// TIA Portal V20 export
FUNCTION_BLOCK "Sequence_1_VisionUnit"   // FB160, LAD
TITLE = Sequence
// Sequence template programmend in ladder logic
// stored: IsIECCheckEnabled true, MemoryReserve 100, Namespace Unit1.Em6, SetENOAutomatically true
   VAR_OUTPUT
      safeState : Bool;
   END_VAR
   VAR
      instSequenceLADControl { ExternalWritable := 'False'} : "LAF_ControlLadSequence";
      instSequenceLADStatus { ExternalWritable := 'False'} : "LAF_StatusLadSequence";
      statPulse { ExternalWritable := 'False'} : Array[0..999] of Bool;
      statTonTimer { ExternalWritable := 'False'} : Array[0..1999] of TON_TIME;
   END_VAR
   VAR_TEMP
      tempCustomerAction : Bool;   // Placeholder for possible actions
      tempDo_nothing_and_wait_for_init : Bool;   // Placeholder for doing nothing
      tempSafeStateCondition : Bool;   // Temp Condition for the equipment module to be in a safe state
   END_VAR
   VAR CONSTANT
      STEP_IDLE : DInt := 1;   // Idle Step
      JOB_1_STEP_01 : DInt := 101;
      JOB_1_STEP_11 : DInt := 111;
      JOB_1_STEP_21 : DInt := 121;
      JOB_1_STEP_31 : DInt := 131;
      JOB_1_STEP_91 : DInt := 191;
      JOB_2_STEP_01 : DInt := 201;
      JOB_2_STEP_11 : DInt := 211;
      JOB_2_STEP_91 : DInt := 291;
      JOB_3_STEP_01 : DInt := 301;
      JOB_3_STEP_11 : DInt := 311;
      JOB_3_STEP_91 : DInt := 391;
      JOB_10_STEP_01 : DInt := 1001;
      JOB_10_STEP_11 : DInt := 1011;
      JOB_10_STEP_21 : DInt := 1021;
      JOB_10_STEP_31 : DInt := 1031;
      JOB_10_STEP_41 : DInt := 1041;
      JOB_10_STEP_51 : DInt := 1051;
      JOB_10_STEP_61 : DInt := 1061;
      JOB_10_STEP_71 : DInt := 1071;
      JOB_10_STEP_81 : DInt := 1081;
      JOB_10_STEP_91 : DInt := 1091;
      STEP_IMMEDIATE_STOP : DInt := 9001;   // Step executed when an immediate stop command is triggered for the sequence (i.e. when unit is in state aborting)
      SeqDelayTime : Time := T#100ms;
      SeqNoDelayTime : Time;
      TRUE : Bool := TRUE;
      FALSE : Bool := FALSE;
      VisionUnitAxisZHomePos : SInt := 0;
      VisionUnitAxisZVisionPos : SInt := 1;
   END_VAR
   VAR_TEMP   // added for the SCL form of the ladder/FBD networks
      _w1 : Bool;
      _w2 : Bool;
   END_VAR
BEGIN

REGION Network 1: BLOCK INFO HEADER
   // (company) / (C) Copyright (year)
   // ---------------------------------------------------------------------------------
   // Title:                             (Title of this block)
   // Comment/Function: (that is implemented in the block)
   // Library/Family:           (that the source is dedicated to)
   // Author:                        (department / person in charge / contact)
   // Target System:          (test system with FW version)
   // Engineering:              TIA Portal (SW version)
   // Restrictions:               (OB types, etc.)
   // Requirements:           (hardware, technological package, etc.)
   // ---------------------------------------------------------------------------------
   // Change log table:
   // Version          | Date             | Signature      | Expert in charge  | Changes applied ------------------------|----------------------|-------------------------|--------------------------------|-----------------------
   // 001.000.000 | yyyy-mm-dd | 0x00000000 | (name of expert) | First released version
END_REGION

REGION Network 2: DESCRIPTION
   // This is a template block provided by the Automation Framework. It can be used to create an own project.
   // The Block Info Header is prepared to put in your own data.
   // Description of the block could be added here and the docu created by Code2Docu.
END_REGION

REGION Network 3: *************** CONTROL **********************
END_REGION

REGION Network 4: Sequence Control
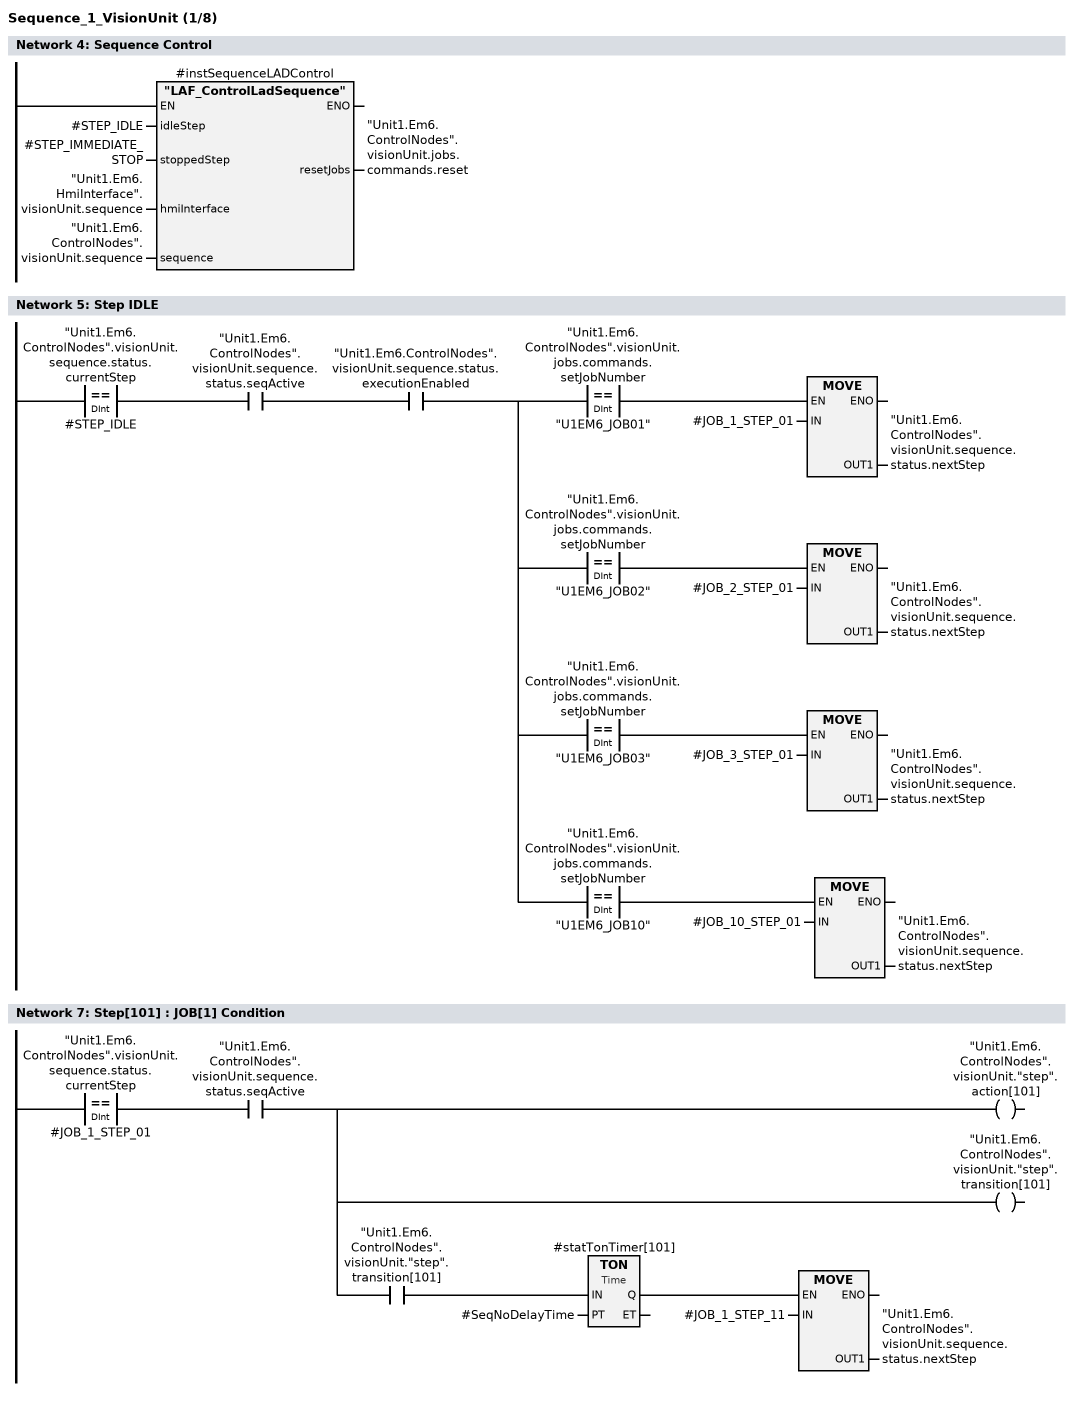
   RUNG wire#powerrail
      #instSequenceLADControl(idleStep := #STEP_IDLE, stoppedStep := #STEP_IMMEDIATE_STOP, hmiInterface := "Unit1.Em6.HmiInterface".visionUnit.sequence, sequence := "Unit1.Em6.ControlNodes".visionUnit.sequence, resetJobs => "Unit1.Em6.ControlNodes".visionUnit.jobs.commands.reset)
   END_RUNG
   // the same network as SCL:
   #instSequenceLADControl(idleStep := #STEP_IDLE,   // "LAF_ControlLadSequence"
                           stoppedStep := #STEP_IMMEDIATE_STOP,
                           hmiInterface := "Unit1.Em6.HmiInterface".visionUnit.sequence,
                           sequence := "Unit1.Em6.ControlNodes".visionUnit.sequence,
                           resetJobs => "Unit1.Em6.ControlNodes".visionUnit.jobs.commands.reset);
END_REGION

REGION Network 5: Step IDLE
   RUNG wire#powerrail
      { S7_Templates := "SrcType := DInt" } EQ_Contact(in1 := "Unit1.Em6.ControlNodes".visionUnit.sequence.status.currentStep, in2 := #STEP_IDLE)
      Contact( "Unit1.Em6.ControlNodes".visionUnit.sequence.status.seqActive )
      Contact( "Unit1.Em6.ControlNodes".visionUnit.sequence.status.executionEnabled )
      wire#w1
      { S7_Templates := "SrcType := DInt" } EQ_Contact(in1 := "Unit1.Em6.ControlNodes".visionUnit.jobs.commands.setJobNumber, in2 := "U1EM6_JOB01")
      Move(in := #JOB_1_STEP_01, out1 => "Unit1.Em6.ControlNodes".visionUnit.sequence.status.nextStep)
   END_RUNG
   RUNG wire#w1
      { S7_Templates := "SrcType := DInt" } EQ_Contact(in1 := "Unit1.Em6.ControlNodes".visionUnit.jobs.commands.setJobNumber, in2 := "U1EM6_JOB02")
      Move(in := #JOB_2_STEP_01, out1 => "Unit1.Em6.ControlNodes".visionUnit.sequence.status.nextStep)
   END_RUNG
   RUNG wire#w1
      { S7_Templates := "SrcType := DInt" } EQ_Contact(in1 := "Unit1.Em6.ControlNodes".visionUnit.jobs.commands.setJobNumber, in2 := "U1EM6_JOB03")
      Move(in := #JOB_3_STEP_01, out1 => "Unit1.Em6.ControlNodes".visionUnit.sequence.status.nextStep)
   END_RUNG
   RUNG wire#w1
      { S7_Templates := "SrcType := DInt" } EQ_Contact(in1 := "Unit1.Em6.ControlNodes".visionUnit.jobs.commands.setJobNumber, in2 := "U1EM6_JOB10")
      Move(in := #JOB_10_STEP_01, out1 => "Unit1.Em6.ControlNodes".visionUnit.sequence.status.nextStep)
   END_RUNG
   // the same network as SCL:
   #_w1 := ("Unit1.Em6.ControlNodes".visionUnit.sequence.status.currentStep = #STEP_IDLE) AND "Unit1.Em6.ControlNodes".visionUnit.sequence.status.seqActive AND "Unit1.Em6.ControlNodes".visionUnit.sequence.status.executionEnabled;
   IF #_w1 AND ("Unit1.Em6.ControlNodes".visionUnit.jobs.commands.setJobNumber = "U1EM6_JOB01") THEN
       "Unit1.Em6.ControlNodes".visionUnit.sequence.status.nextStep := #JOB_1_STEP_01;
   END_IF;
   IF #_w1 AND ("Unit1.Em6.ControlNodes".visionUnit.jobs.commands.setJobNumber = "U1EM6_JOB02") THEN
       "Unit1.Em6.ControlNodes".visionUnit.sequence.status.nextStep := #JOB_2_STEP_01;
   END_IF;
   IF #_w1 AND ("Unit1.Em6.ControlNodes".visionUnit.jobs.commands.setJobNumber = "U1EM6_JOB03") THEN
       "Unit1.Em6.ControlNodes".visionUnit.sequence.status.nextStep := #JOB_3_STEP_01;
   END_IF;
   IF #_w1 AND ("Unit1.Em6.ControlNodes".visionUnit.jobs.commands.setJobNumber = "U1EM6_JOB10") THEN
       "Unit1.Em6.ControlNodes".visionUnit.sequence.status.nextStep := #JOB_10_STEP_01;
   END_IF;
END_REGION

REGION Network 6: *************** JOB 1 EM READY *************************
END_REGION

REGION Network 7: Step[101] : JOB[1] Condition
   RUNG wire#powerrail
      { S7_Templates := "SrcType := DInt" } EQ_Contact(in1 := "Unit1.Em6.ControlNodes".visionUnit.sequence.status.currentStep, in2 := #JOB_1_STEP_01)
      Contact( "Unit1.Em6.ControlNodes".visionUnit.sequence.status.seqActive )
      wire#w1
      Coil( "Unit1.Em6.ControlNodes".visionUnit."step".action[101] )
   END_RUNG
   RUNG wire#w1
      Coil( "Unit1.Em6.ControlNodes".visionUnit."step".transition[101] )
   END_RUNG
   RUNG wire#w1
      Contact( "Unit1.Em6.ControlNodes".visionUnit."step".transition[101] )
      { S7_Templates := "time_type := Time" } #statTonTimer[101].TON(pt := #SeqNoDelayTime, et =>)
      Move(in := #JOB_1_STEP_11, out1 => "Unit1.Em6.ControlNodes".visionUnit.sequence.status.nextStep)
   END_RUNG
   // the same network as SCL:
   "Unit1.Em6.ControlNodes".visionUnit."step".action[101] := ("Unit1.Em6.ControlNodes".visionUnit.sequence.status.currentStep = #JOB_1_STEP_01) AND "Unit1.Em6.ControlNodes".visionUnit.sequence.status.seqActive;
   "Unit1.Em6.ControlNodes".visionUnit."step".transition[101] := ("Unit1.Em6.ControlNodes".visionUnit.sequence.status.currentStep = #JOB_1_STEP_01) AND "Unit1.Em6.ControlNodes".visionUnit.sequence.status.seqActive;
   #statTonTimer[101].TON(IN := ("Unit1.Em6.ControlNodes".visionUnit.sequence.status.currentStep = #JOB_1_STEP_01) AND "Unit1.Em6.ControlNodes".visionUnit.sequence.status.seqActive AND "Unit1.Em6.ControlNodes".visionUnit."step".transition[101],
                          PT := #SeqNoDelayTime);
   IF #statTonTimer[101].Q THEN
       "Unit1.Em6.ControlNodes".visionUnit.sequence.status.nextStep := #JOB_1_STEP_11;
   END_IF;
END_REGION

REGION Network 8: Step[111] : Vision Unit AxisZ Homed Check
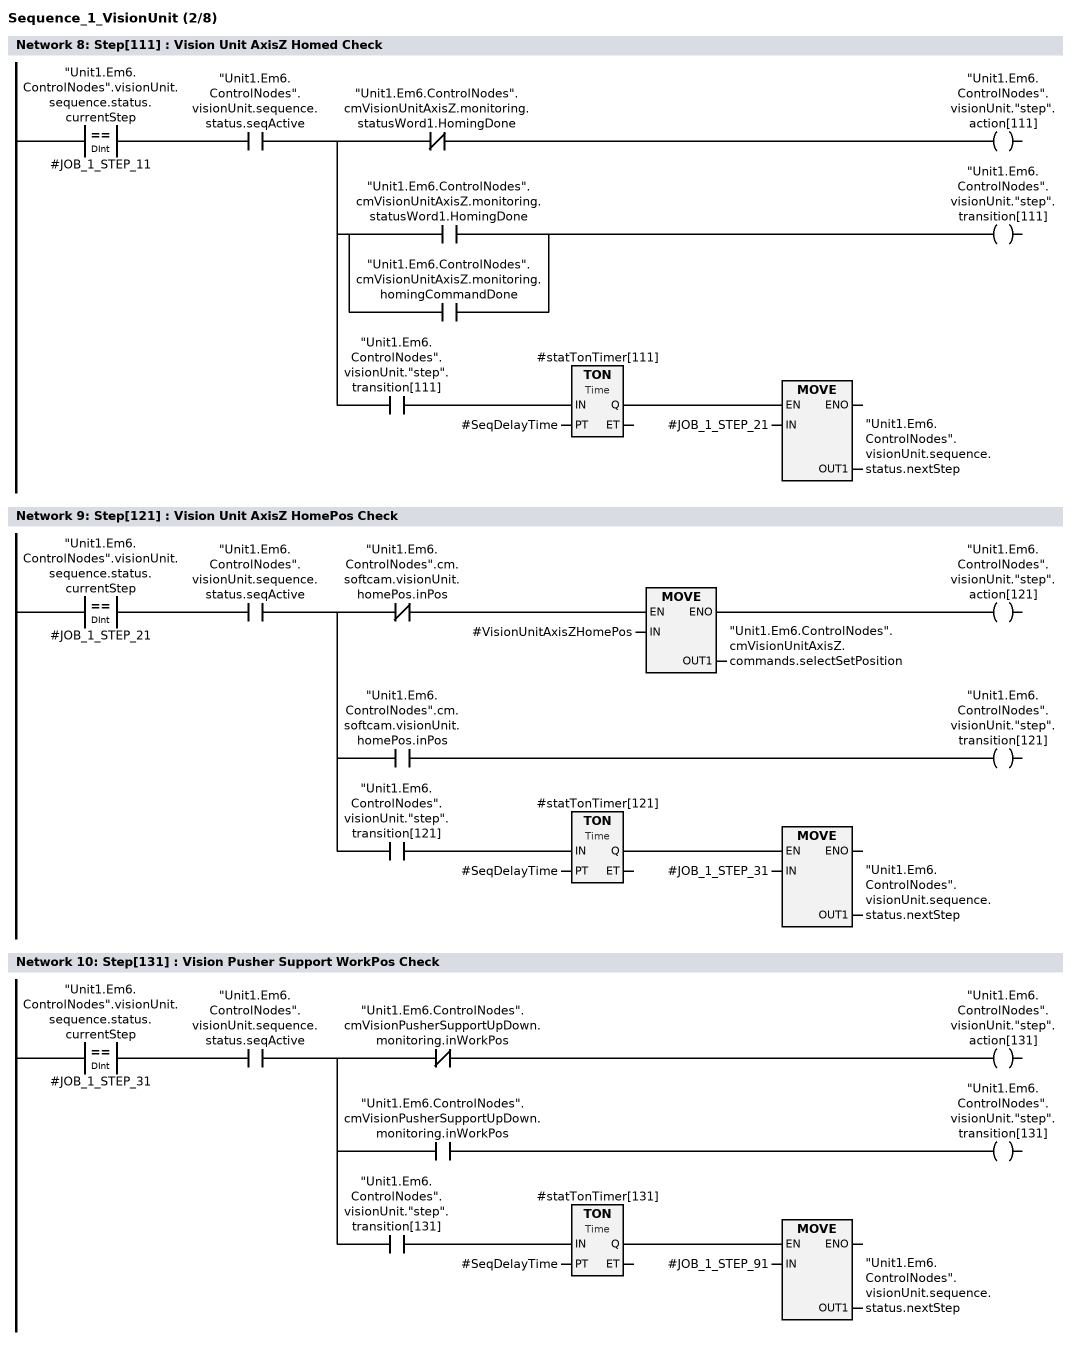
   RUNG wire#powerrail
      { S7_Templates := "SrcType := DInt" } EQ_Contact(in1 := "Unit1.Em6.ControlNodes".visionUnit.sequence.status.currentStep, in2 := #JOB_1_STEP_11)
      Contact( "Unit1.Em6.ControlNodes".visionUnit.sequence.status.seqActive )
      wire#w1
      I_Contact( "Unit1.Em6.ControlNodes".cmVisionUnitAxisZ.monitoring.statusWord1.HomingDone )
      Coil( "Unit1.Em6.ControlNodes".visionUnit."step".action[111] )
   END_RUNG
   RUNG wire#w1
      Contact( "Unit1.Em6.ControlNodes".cmVisionUnitAxisZ.monitoring.statusWord1.HomingDone )
      wire#w2
      Coil( "Unit1.Em6.ControlNodes".visionUnit."step".transition[111] )
   END_RUNG
   RUNG wire#w1
      Contact( "Unit1.Em6.ControlNodes".cmVisionUnitAxisZ.monitoring.homingCommandDone )
   END_RUNG wire#w2
   RUNG wire#w1
      Contact( "Unit1.Em6.ControlNodes".visionUnit."step".transition[111] )
      { S7_Templates := "time_type := Time" } #statTonTimer[111].TON(pt := #SeqDelayTime, et =>)
      Move(in := #JOB_1_STEP_21, out1 => "Unit1.Em6.ControlNodes".visionUnit.sequence.status.nextStep)
   END_RUNG
   // the same network as SCL:
   #_w1 := ("Unit1.Em6.ControlNodes".visionUnit.sequence.status.currentStep = #JOB_1_STEP_11) AND "Unit1.Em6.ControlNodes".visionUnit.sequence.status.seqActive;
   "Unit1.Em6.ControlNodes".visionUnit."step".action[111] := #_w1 AND NOT "Unit1.Em6.ControlNodes".cmVisionUnitAxisZ.monitoring.statusWord1.HomingDone;
   "Unit1.Em6.ControlNodes".visionUnit."step".transition[111] := #_w1 AND ("Unit1.Em6.ControlNodes".cmVisionUnitAxisZ.monitoring.statusWord1.HomingDone OR "Unit1.Em6.ControlNodes".cmVisionUnitAxisZ.monitoring.homingCommandDone);
   #statTonTimer[111].TON(IN := #_w1 AND "Unit1.Em6.ControlNodes".visionUnit."step".transition[111],
                          PT := #SeqDelayTime);
   IF #statTonTimer[111].Q THEN
       "Unit1.Em6.ControlNodes".visionUnit.sequence.status.nextStep := #JOB_1_STEP_21;
   END_IF;
END_REGION

REGION Network 9: Step[121] : Vision Unit AxisZ HomePos Check
   RUNG wire#powerrail
      { S7_Templates := "SrcType := DInt" } EQ_Contact(in1 := "Unit1.Em6.ControlNodes".visionUnit.sequence.status.currentStep, in2 := #JOB_1_STEP_21)
      Contact( "Unit1.Em6.ControlNodes".visionUnit.sequence.status.seqActive )
      wire#w1
      I_Contact( "Unit1.Em6.ControlNodes".cm.softcam.visionUnit.homePos.inPos )
      Move(in := #VisionUnitAxisZHomePos, out1 => "Unit1.Em6.ControlNodes".cmVisionUnitAxisZ.commands.selectSetPosition)
      Coil( "Unit1.Em6.ControlNodes".visionUnit."step".action[121] )
   END_RUNG
   RUNG wire#w1
      Contact( "Unit1.Em6.ControlNodes".cm.softcam.visionUnit.homePos.inPos )
      Coil( "Unit1.Em6.ControlNodes".visionUnit."step".transition[121] )
   END_RUNG
   RUNG wire#w1
      Contact( "Unit1.Em6.ControlNodes".visionUnit."step".transition[121] )
      { S7_Templates := "time_type := Time" } #statTonTimer[121].TON(pt := #SeqDelayTime, et =>)
      Move(in := #JOB_1_STEP_31, out1 => "Unit1.Em6.ControlNodes".visionUnit.sequence.status.nextStep)
   END_RUNG
   // the same network as SCL:
   #_w1 := ("Unit1.Em6.ControlNodes".visionUnit.sequence.status.currentStep = #JOB_1_STEP_21) AND "Unit1.Em6.ControlNodes".visionUnit.sequence.status.seqActive;
   #_w2 := #_w1 AND NOT "Unit1.Em6.ControlNodes".cm.softcam.visionUnit.homePos.inPos;
   IF #_w2 THEN
       "Unit1.Em6.ControlNodes".cmVisionUnitAxisZ.commands.selectSetPosition := #VisionUnitAxisZHomePos;
   END_IF;
   "Unit1.Em6.ControlNodes".visionUnit."step".action[121] := #_w2;
   "Unit1.Em6.ControlNodes".visionUnit."step".transition[121] := #_w1 AND "Unit1.Em6.ControlNodes".cm.softcam.visionUnit.homePos.inPos;
   #statTonTimer[121].TON(IN := #_w1 AND "Unit1.Em6.ControlNodes".visionUnit."step".transition[121],
                          PT := #SeqDelayTime);
   IF #statTonTimer[121].Q THEN
       "Unit1.Em6.ControlNodes".visionUnit.sequence.status.nextStep := #JOB_1_STEP_31;
   END_IF;
END_REGION

REGION Network 10: Step[131] : Vision Pusher Support WorkPos Check
   RUNG wire#powerrail
      { S7_Templates := "SrcType := DInt" } EQ_Contact(in1 := "Unit1.Em6.ControlNodes".visionUnit.sequence.status.currentStep, in2 := #JOB_1_STEP_31)
      Contact( "Unit1.Em6.ControlNodes".visionUnit.sequence.status.seqActive )
      wire#w1
      I_Contact( "Unit1.Em6.ControlNodes".cmVisionPusherSupportUpDown.monitoring.inWorkPos )
      Coil( "Unit1.Em6.ControlNodes".visionUnit."step".action[131] )
   END_RUNG
   RUNG wire#w1
      Contact( "Unit1.Em6.ControlNodes".cmVisionPusherSupportUpDown.monitoring.inWorkPos )
      Coil( "Unit1.Em6.ControlNodes".visionUnit."step".transition[131] )
   END_RUNG
   RUNG wire#w1
      Contact( "Unit1.Em6.ControlNodes".visionUnit."step".transition[131] )
      { S7_Templates := "time_type := Time" } #statTonTimer[131].TON(pt := #SeqDelayTime, et =>)
      Move(in := #JOB_1_STEP_91, out1 => "Unit1.Em6.ControlNodes".visionUnit.sequence.status.nextStep)
   END_RUNG
   // the same network as SCL:
   #_w1 := ("Unit1.Em6.ControlNodes".visionUnit.sequence.status.currentStep = #JOB_1_STEP_31) AND "Unit1.Em6.ControlNodes".visionUnit.sequence.status.seqActive;
   "Unit1.Em6.ControlNodes".visionUnit."step".action[131] := #_w1 AND NOT "Unit1.Em6.ControlNodes".cmVisionPusherSupportUpDown.monitoring.inWorkPos;
   "Unit1.Em6.ControlNodes".visionUnit."step".transition[131] := #_w1 AND "Unit1.Em6.ControlNodes".cmVisionPusherSupportUpDown.monitoring.inWorkPos;
   #statTonTimer[131].TON(IN := #_w1 AND "Unit1.Em6.ControlNodes".visionUnit."step".transition[131],
                          PT := #SeqDelayTime);
   IF #statTonTimer[131].Q THEN
       "Unit1.Em6.ControlNodes".visionUnit.sequence.status.nextStep := #JOB_1_STEP_91;
   END_IF;
END_REGION

REGION Network 11: Step[191] : JOB[1] Step End
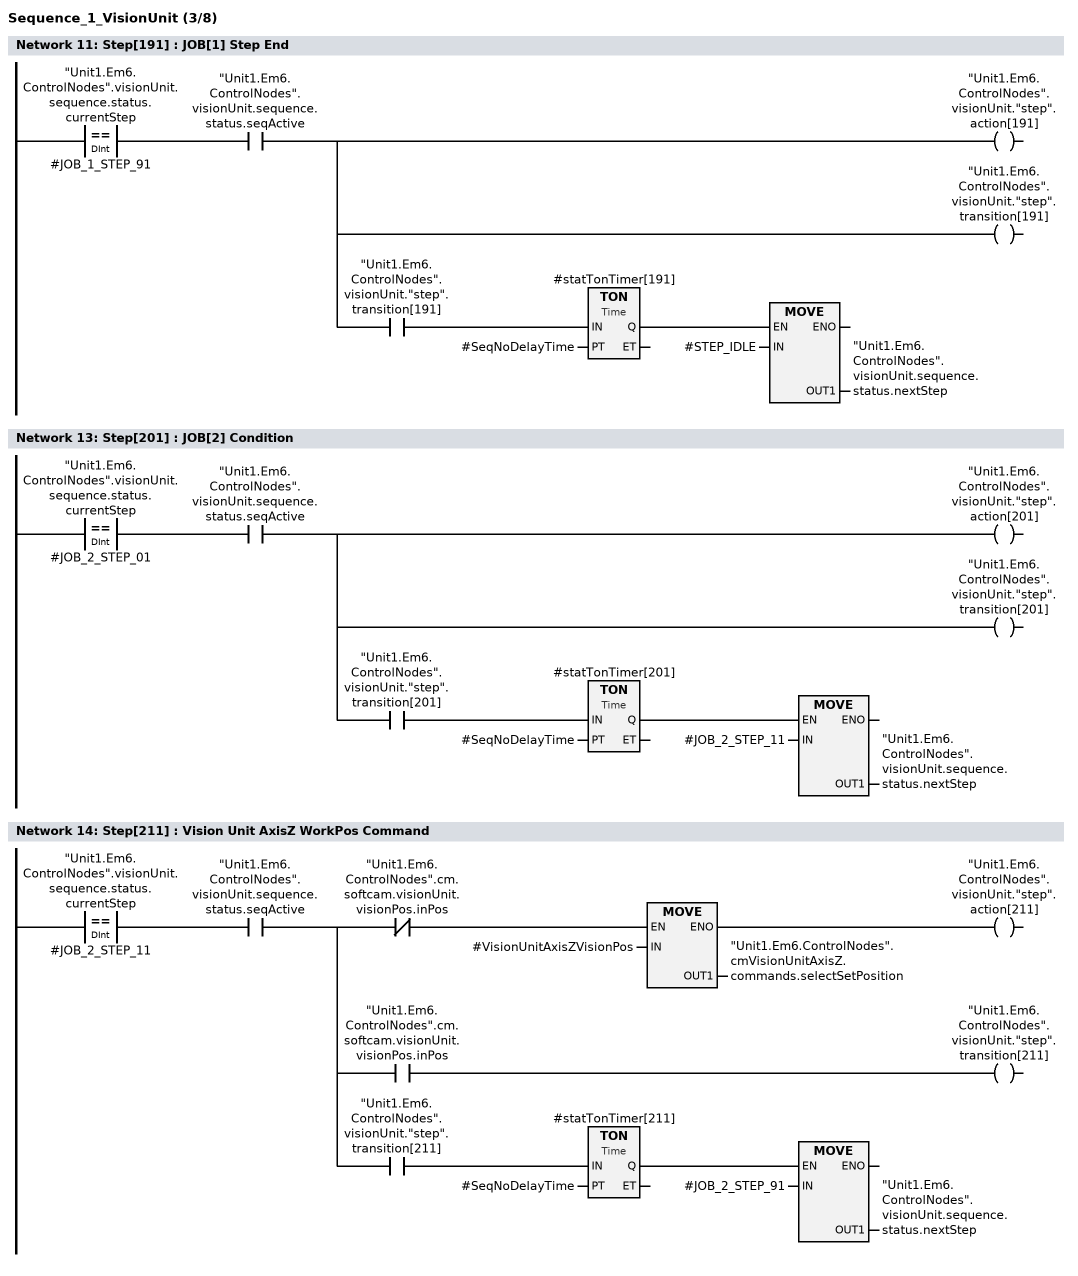
   RUNG wire#powerrail
      { S7_Templates := "SrcType := DInt" } EQ_Contact(in1 := "Unit1.Em6.ControlNodes".visionUnit.sequence.status.currentStep, in2 := #JOB_1_STEP_91)
      Contact( "Unit1.Em6.ControlNodes".visionUnit.sequence.status.seqActive )
      wire#w1
      Coil( "Unit1.Em6.ControlNodes".visionUnit."step".action[191] )
   END_RUNG
   RUNG wire#w1
      Coil( "Unit1.Em6.ControlNodes".visionUnit."step".transition[191] )
   END_RUNG
   RUNG wire#w1
      Contact( "Unit1.Em6.ControlNodes".visionUnit."step".transition[191] )
      { S7_Templates := "time_type := Time" } #statTonTimer[191].TON(pt := #SeqNoDelayTime, et =>)
      Move(in := #STEP_IDLE, out1 => "Unit1.Em6.ControlNodes".visionUnit.sequence.status.nextStep)
   END_RUNG
   // the same network as SCL:
   "Unit1.Em6.ControlNodes".visionUnit."step".action[191] := ("Unit1.Em6.ControlNodes".visionUnit.sequence.status.currentStep = #JOB_1_STEP_91) AND "Unit1.Em6.ControlNodes".visionUnit.sequence.status.seqActive;
   "Unit1.Em6.ControlNodes".visionUnit."step".transition[191] := ("Unit1.Em6.ControlNodes".visionUnit.sequence.status.currentStep = #JOB_1_STEP_91) AND "Unit1.Em6.ControlNodes".visionUnit.sequence.status.seqActive;
   #statTonTimer[191].TON(IN := ("Unit1.Em6.ControlNodes".visionUnit.sequence.status.currentStep = #JOB_1_STEP_91) AND "Unit1.Em6.ControlNodes".visionUnit.sequence.status.seqActive AND "Unit1.Em6.ControlNodes".visionUnit."step".transition[191],
                          PT := #SeqNoDelayTime);
   IF #statTonTimer[191].Q THEN
       "Unit1.Em6.ControlNodes".visionUnit.sequence.status.nextStep := #STEP_IDLE;
   END_IF;
END_REGION

REGION Network 12: *************** JOB 2 VISION UNIT DOWN AUTO *************************
END_REGION

REGION Network 13: Step[201] : JOB[2] Condition
   RUNG wire#powerrail
      { S7_Templates := "SrcType := DInt" } EQ_Contact(in1 := "Unit1.Em6.ControlNodes".visionUnit.sequence.status.currentStep, in2 := #JOB_2_STEP_01)
      Contact( "Unit1.Em6.ControlNodes".visionUnit.sequence.status.seqActive )
      wire#w1
      Coil( "Unit1.Em6.ControlNodes".visionUnit."step".action[201] )
   END_RUNG
   RUNG wire#w1
      Coil( "Unit1.Em6.ControlNodes".visionUnit."step".transition[201] )
   END_RUNG
   RUNG wire#w1
      Contact( "Unit1.Em6.ControlNodes".visionUnit."step".transition[201] )
      { S7_Templates := "time_type := Time" } #statTonTimer[201].TON(pt := #SeqNoDelayTime, et =>)
      Move(in := #JOB_2_STEP_11, out1 => "Unit1.Em6.ControlNodes".visionUnit.sequence.status.nextStep)
   END_RUNG
   // the same network as SCL:
   "Unit1.Em6.ControlNodes".visionUnit."step".action[201] := ("Unit1.Em6.ControlNodes".visionUnit.sequence.status.currentStep = #JOB_2_STEP_01) AND "Unit1.Em6.ControlNodes".visionUnit.sequence.status.seqActive;
   "Unit1.Em6.ControlNodes".visionUnit."step".transition[201] := ("Unit1.Em6.ControlNodes".visionUnit.sequence.status.currentStep = #JOB_2_STEP_01) AND "Unit1.Em6.ControlNodes".visionUnit.sequence.status.seqActive;
   #statTonTimer[201].TON(IN := ("Unit1.Em6.ControlNodes".visionUnit.sequence.status.currentStep = #JOB_2_STEP_01) AND "Unit1.Em6.ControlNodes".visionUnit.sequence.status.seqActive AND "Unit1.Em6.ControlNodes".visionUnit."step".transition[201],
                          PT := #SeqNoDelayTime);
   IF #statTonTimer[201].Q THEN
       "Unit1.Em6.ControlNodes".visionUnit.sequence.status.nextStep := #JOB_2_STEP_11;
   END_IF;
END_REGION

REGION Network 14: Step[211] : Vision Unit AxisZ WorkPos Command
   RUNG wire#powerrail
      { S7_Templates := "SrcType := DInt" } EQ_Contact(in1 := "Unit1.Em6.ControlNodes".visionUnit.sequence.status.currentStep, in2 := #JOB_2_STEP_11)
      Contact( "Unit1.Em6.ControlNodes".visionUnit.sequence.status.seqActive )
      wire#w1
      I_Contact( "Unit1.Em6.ControlNodes".cm.softcam.visionUnit.visionPos.inPos )
      Move(in := #VisionUnitAxisZVisionPos, out1 => "Unit1.Em6.ControlNodes".cmVisionUnitAxisZ.commands.selectSetPosition)
      Coil( "Unit1.Em6.ControlNodes".visionUnit."step".action[211] )
   END_RUNG
   RUNG wire#w1
      Contact( "Unit1.Em6.ControlNodes".cm.softcam.visionUnit.visionPos.inPos )
      Coil( "Unit1.Em6.ControlNodes".visionUnit."step".transition[211] )
   END_RUNG
   RUNG wire#w1
      Contact( "Unit1.Em6.ControlNodes".visionUnit."step".transition[211] )
      { S7_Templates := "time_type := Time" } #statTonTimer[211].TON(pt := #SeqNoDelayTime, et =>)
      Move(in := #JOB_2_STEP_91, out1 => "Unit1.Em6.ControlNodes".visionUnit.sequence.status.nextStep)
   END_RUNG
   // the same network as SCL:
   #_w1 := ("Unit1.Em6.ControlNodes".visionUnit.sequence.status.currentStep = #JOB_2_STEP_11) AND "Unit1.Em6.ControlNodes".visionUnit.sequence.status.seqActive;
   #_w2 := #_w1 AND NOT "Unit1.Em6.ControlNodes".cm.softcam.visionUnit.visionPos.inPos;
   IF #_w2 THEN
       "Unit1.Em6.ControlNodes".cmVisionUnitAxisZ.commands.selectSetPosition := #VisionUnitAxisZVisionPos;
   END_IF;
   "Unit1.Em6.ControlNodes".visionUnit."step".action[211] := #_w2;
   "Unit1.Em6.ControlNodes".visionUnit."step".transition[211] := #_w1 AND "Unit1.Em6.ControlNodes".cm.softcam.visionUnit.visionPos.inPos;
   #statTonTimer[211].TON(IN := #_w1 AND "Unit1.Em6.ControlNodes".visionUnit."step".transition[211],
                          PT := #SeqNoDelayTime);
   IF #statTonTimer[211].Q THEN
       "Unit1.Em6.ControlNodes".visionUnit.sequence.status.nextStep := #JOB_2_STEP_91;
   END_IF;
END_REGION

REGION Network 15: Step[291] : JOB[2] Step End
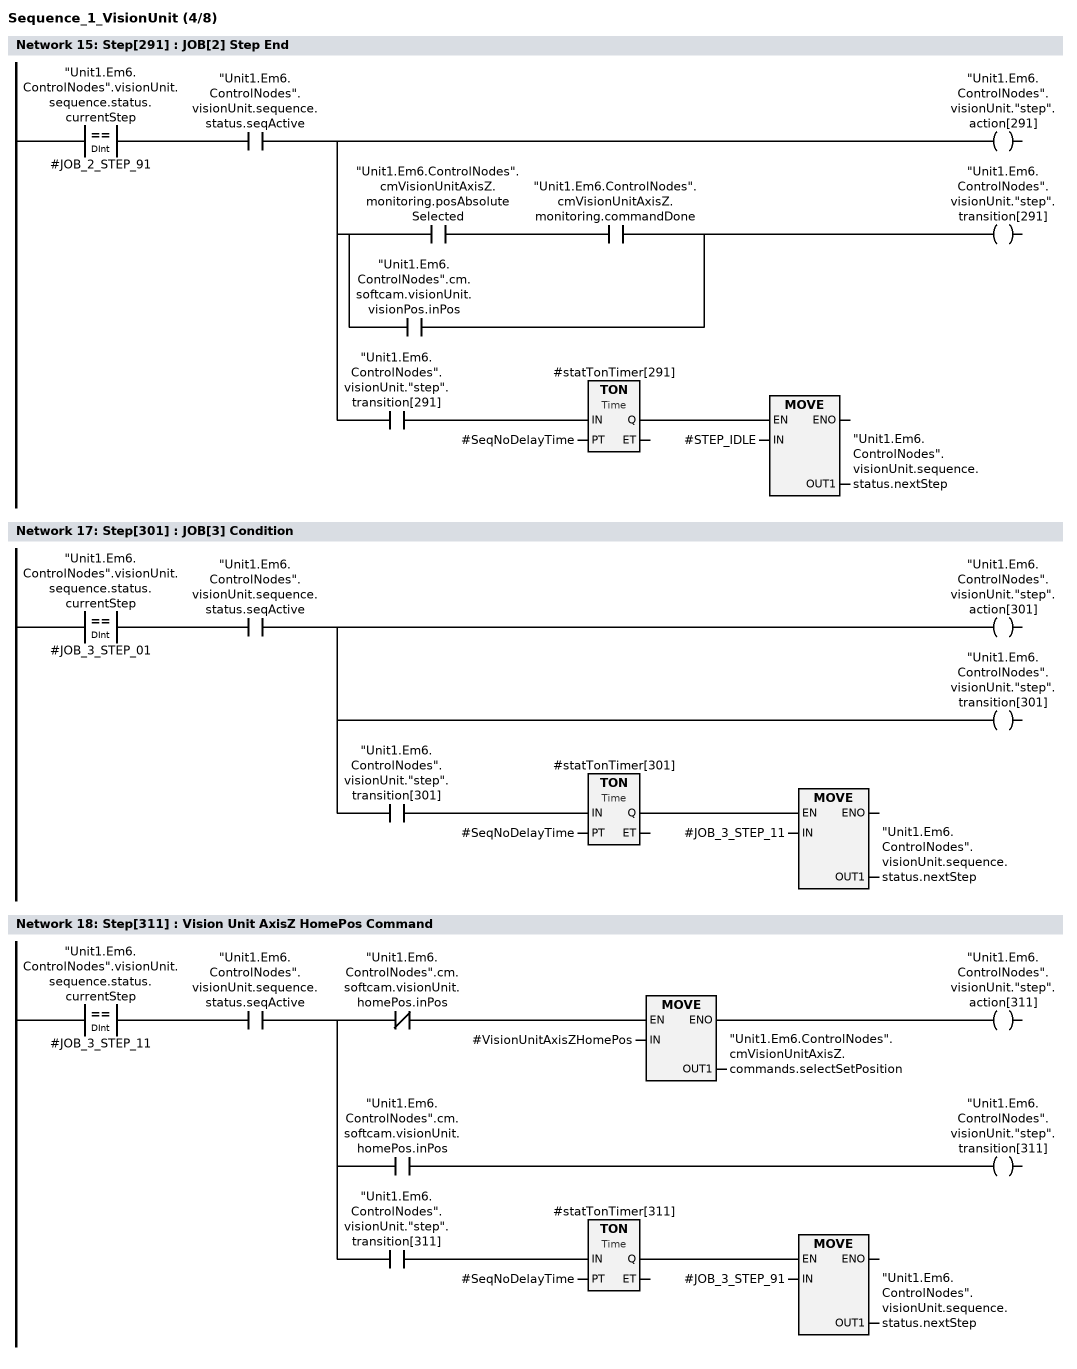
   RUNG wire#powerrail
      { S7_Templates := "SrcType := DInt" } EQ_Contact(in1 := "Unit1.Em6.ControlNodes".visionUnit.sequence.status.currentStep, in2 := #JOB_2_STEP_91)
      Contact( "Unit1.Em6.ControlNodes".visionUnit.sequence.status.seqActive )
      wire#w1
      Coil( "Unit1.Em6.ControlNodes".visionUnit."step".action[291] )
   END_RUNG
   RUNG wire#w1
      Contact( "Unit1.Em6.ControlNodes".cmVisionUnitAxisZ.monitoring.posAbsoluteSelected )
      Contact( "Unit1.Em6.ControlNodes".cmVisionUnitAxisZ.monitoring.commandDone )
      wire#w2
      Coil( "Unit1.Em6.ControlNodes".visionUnit."step".transition[291] )
   END_RUNG
   RUNG wire#w1
      Contact( "Unit1.Em6.ControlNodes".cm.softcam.visionUnit.visionPos.inPos )
   END_RUNG wire#w2
   RUNG wire#w1
      Contact( "Unit1.Em6.ControlNodes".visionUnit."step".transition[291] )
      { S7_Templates := "time_type := Time" } #statTonTimer[291].TON(pt := #SeqNoDelayTime, et =>)
      Move(in := #STEP_IDLE, out1 => "Unit1.Em6.ControlNodes".visionUnit.sequence.status.nextStep)
   END_RUNG
   // the same network as SCL:
   "Unit1.Em6.ControlNodes".visionUnit."step".action[291] := ("Unit1.Em6.ControlNodes".visionUnit.sequence.status.currentStep = #JOB_2_STEP_91) AND "Unit1.Em6.ControlNodes".visionUnit.sequence.status.seqActive;
   "Unit1.Em6.ControlNodes".visionUnit."step".transition[291] := ("Unit1.Em6.ControlNodes".visionUnit.sequence.status.currentStep = #JOB_2_STEP_91) AND "Unit1.Em6.ControlNodes".visionUnit.sequence.status.seqActive AND (("Unit1.Em6.ControlNodes".cmVisionUnitAxisZ.monitoring.posAbsoluteSelected AND "Unit1.Em6.ControlNodes".cmVisionUnitAxisZ.monitoring.commandDone) OR "Unit1.Em6.ControlNodes".cm.softcam.visionUnit.visionPos.inPos);
   #statTonTimer[291].TON(IN := ("Unit1.Em6.ControlNodes".visionUnit.sequence.status.currentStep = #JOB_2_STEP_91) AND "Unit1.Em6.ControlNodes".visionUnit.sequence.status.seqActive AND "Unit1.Em6.ControlNodes".visionUnit."step".transition[291],
                          PT := #SeqNoDelayTime);
   IF #statTonTimer[291].Q THEN
       "Unit1.Em6.ControlNodes".visionUnit.sequence.status.nextStep := #STEP_IDLE;
   END_IF;
END_REGION

REGION Network 16: *************** JOB 3 VISION UNIT UP AUTO *************************
END_REGION

REGION Network 17: Step[301] : JOB[3] Condition
   RUNG wire#powerrail
      { S7_Templates := "SrcType := DInt" } EQ_Contact(in1 := "Unit1.Em6.ControlNodes".visionUnit.sequence.status.currentStep, in2 := #JOB_3_STEP_01)
      Contact( "Unit1.Em6.ControlNodes".visionUnit.sequence.status.seqActive )
      wire#w1
      Coil( "Unit1.Em6.ControlNodes".visionUnit."step".action[301] )
   END_RUNG
   RUNG wire#w1
      Coil( "Unit1.Em6.ControlNodes".visionUnit."step".transition[301] )
   END_RUNG
   RUNG wire#w1
      Contact( "Unit1.Em6.ControlNodes".visionUnit."step".transition[301] )
      { S7_Templates := "time_type := Time" } #statTonTimer[301].TON(pt := #SeqNoDelayTime, et =>)
      Move(in := #JOB_3_STEP_11, out1 => "Unit1.Em6.ControlNodes".visionUnit.sequence.status.nextStep)
   END_RUNG
   // the same network as SCL:
   "Unit1.Em6.ControlNodes".visionUnit."step".action[301] := ("Unit1.Em6.ControlNodes".visionUnit.sequence.status.currentStep = #JOB_3_STEP_01) AND "Unit1.Em6.ControlNodes".visionUnit.sequence.status.seqActive;
   "Unit1.Em6.ControlNodes".visionUnit."step".transition[301] := ("Unit1.Em6.ControlNodes".visionUnit.sequence.status.currentStep = #JOB_3_STEP_01) AND "Unit1.Em6.ControlNodes".visionUnit.sequence.status.seqActive;
   #statTonTimer[301].TON(IN := ("Unit1.Em6.ControlNodes".visionUnit.sequence.status.currentStep = #JOB_3_STEP_01) AND "Unit1.Em6.ControlNodes".visionUnit.sequence.status.seqActive AND "Unit1.Em6.ControlNodes".visionUnit."step".transition[301],
                          PT := #SeqNoDelayTime);
   IF #statTonTimer[301].Q THEN
       "Unit1.Em6.ControlNodes".visionUnit.sequence.status.nextStep := #JOB_3_STEP_11;
   END_IF;
END_REGION

REGION Network 18: Step[311] : Vision Unit AxisZ HomePos Command
   RUNG wire#powerrail
      { S7_Templates := "SrcType := DInt" } EQ_Contact(in1 := "Unit1.Em6.ControlNodes".visionUnit.sequence.status.currentStep, in2 := #JOB_3_STEP_11)
      Contact( "Unit1.Em6.ControlNodes".visionUnit.sequence.status.seqActive )
      wire#w1
      I_Contact( "Unit1.Em6.ControlNodes".cm.softcam.visionUnit.homePos.inPos )
      Move(in := #VisionUnitAxisZHomePos, out1 => "Unit1.Em6.ControlNodes".cmVisionUnitAxisZ.commands.selectSetPosition)
      Coil( "Unit1.Em6.ControlNodes".visionUnit."step".action[311] )
   END_RUNG
   RUNG wire#w1
      Contact( "Unit1.Em6.ControlNodes".cm.softcam.visionUnit.homePos.inPos )
      Coil( "Unit1.Em6.ControlNodes".visionUnit."step".transition[311] )
   END_RUNG
   RUNG wire#w1
      Contact( "Unit1.Em6.ControlNodes".visionUnit."step".transition[311] )
      { S7_Templates := "time_type := Time" } #statTonTimer[311].TON(pt := #SeqNoDelayTime, et =>)
      Move(in := #JOB_3_STEP_91, out1 => "Unit1.Em6.ControlNodes".visionUnit.sequence.status.nextStep)
   END_RUNG
   // the same network as SCL:
   #_w1 := ("Unit1.Em6.ControlNodes".visionUnit.sequence.status.currentStep = #JOB_3_STEP_11) AND "Unit1.Em6.ControlNodes".visionUnit.sequence.status.seqActive;
   #_w2 := #_w1 AND NOT "Unit1.Em6.ControlNodes".cm.softcam.visionUnit.homePos.inPos;
   IF #_w2 THEN
       "Unit1.Em6.ControlNodes".cmVisionUnitAxisZ.commands.selectSetPosition := #VisionUnitAxisZHomePos;
   END_IF;
   "Unit1.Em6.ControlNodes".visionUnit."step".action[311] := #_w2;
   "Unit1.Em6.ControlNodes".visionUnit."step".transition[311] := #_w1 AND "Unit1.Em6.ControlNodes".cm.softcam.visionUnit.homePos.inPos;
   #statTonTimer[311].TON(IN := #_w1 AND "Unit1.Em6.ControlNodes".visionUnit."step".transition[311],
                          PT := #SeqNoDelayTime);
   IF #statTonTimer[311].Q THEN
       "Unit1.Em6.ControlNodes".visionUnit.sequence.status.nextStep := #JOB_3_STEP_91;
   END_IF;
END_REGION

REGION Network 19: Step[391] : JOB[3] Step End
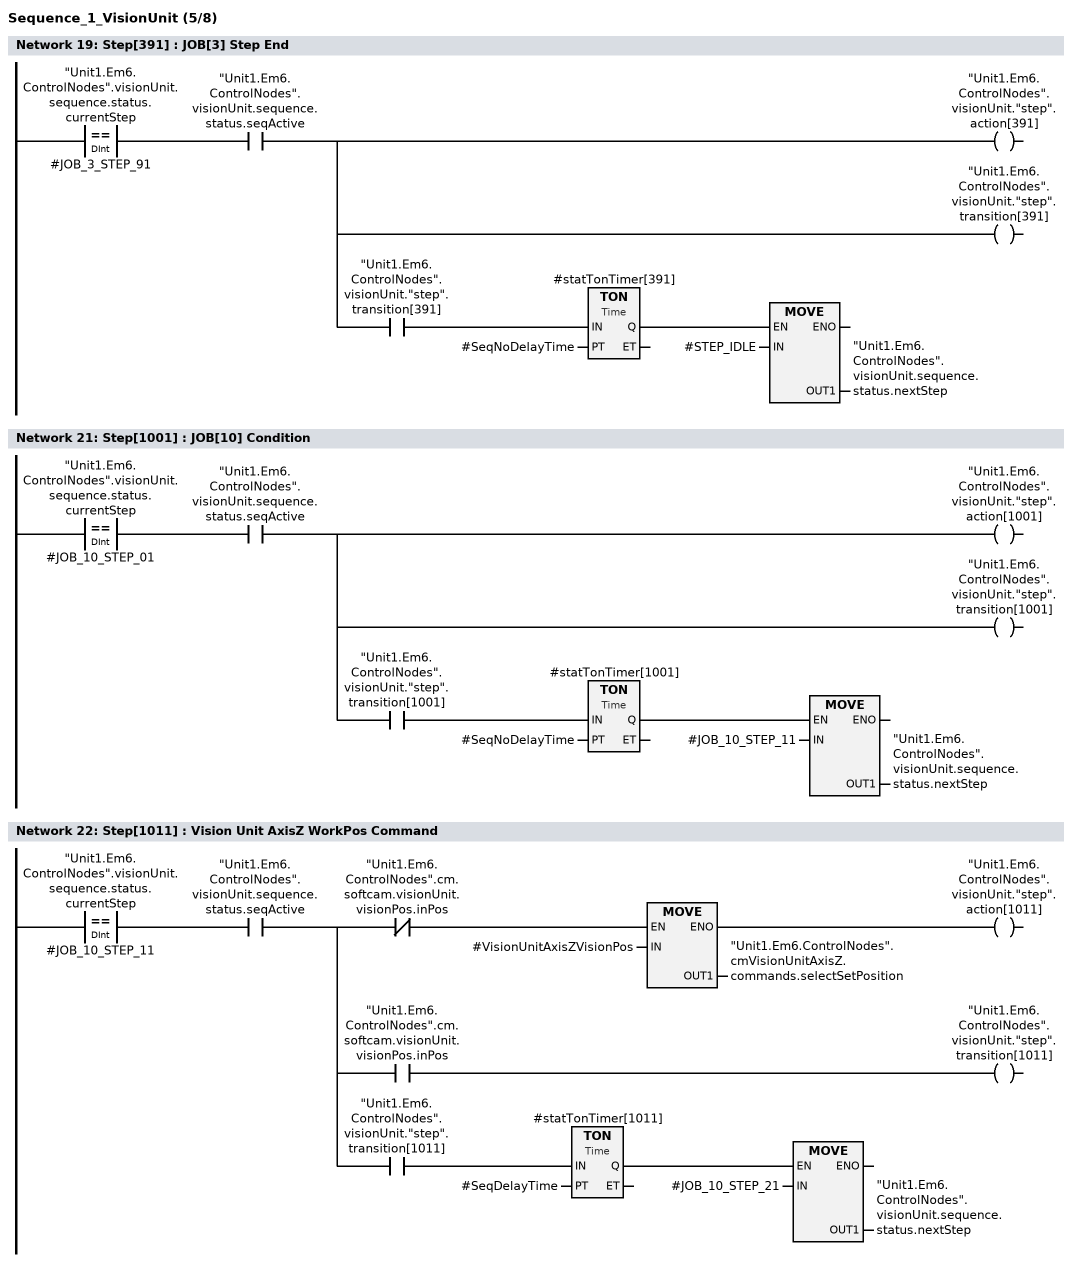
   RUNG wire#powerrail
      { S7_Templates := "SrcType := DInt" } EQ_Contact(in1 := "Unit1.Em6.ControlNodes".visionUnit.sequence.status.currentStep, in2 := #JOB_3_STEP_91)
      Contact( "Unit1.Em6.ControlNodes".visionUnit.sequence.status.seqActive )
      wire#w1
      Coil( "Unit1.Em6.ControlNodes".visionUnit."step".action[391] )
   END_RUNG
   RUNG wire#w1
      Coil( "Unit1.Em6.ControlNodes".visionUnit."step".transition[391] )
   END_RUNG
   RUNG wire#w1
      Contact( "Unit1.Em6.ControlNodes".visionUnit."step".transition[391] )
      { S7_Templates := "time_type := Time" } #statTonTimer[391].TON(pt := #SeqNoDelayTime, et =>)
      Move(in := #STEP_IDLE, out1 => "Unit1.Em6.ControlNodes".visionUnit.sequence.status.nextStep)
   END_RUNG
   // the same network as SCL:
   "Unit1.Em6.ControlNodes".visionUnit."step".action[391] := ("Unit1.Em6.ControlNodes".visionUnit.sequence.status.currentStep = #JOB_3_STEP_91) AND "Unit1.Em6.ControlNodes".visionUnit.sequence.status.seqActive;
   "Unit1.Em6.ControlNodes".visionUnit."step".transition[391] := ("Unit1.Em6.ControlNodes".visionUnit.sequence.status.currentStep = #JOB_3_STEP_91) AND "Unit1.Em6.ControlNodes".visionUnit.sequence.status.seqActive;
   #statTonTimer[391].TON(IN := ("Unit1.Em6.ControlNodes".visionUnit.sequence.status.currentStep = #JOB_3_STEP_91) AND "Unit1.Em6.ControlNodes".visionUnit.sequence.status.seqActive AND "Unit1.Em6.ControlNodes".visionUnit."step".transition[391],
                          PT := #SeqNoDelayTime);
   IF #statTonTimer[391].Q THEN
       "Unit1.Em6.ControlNodes".visionUnit.sequence.status.nextStep := #STEP_IDLE;
   END_IF;
END_REGION

REGION Network 20: *************** JOB 10 VISION FULL AUTO *************************
END_REGION

REGION Network 21: Step[1001] : JOB[10] Condition
   RUNG wire#powerrail
      { S7_Templates := "SrcType := DInt" } EQ_Contact(in1 := "Unit1.Em6.ControlNodes".visionUnit.sequence.status.currentStep, in2 := #JOB_10_STEP_01)
      Contact( "Unit1.Em6.ControlNodes".visionUnit.sequence.status.seqActive )
      wire#w1
      Coil( "Unit1.Em6.ControlNodes".visionUnit."step".action[1001] )
   END_RUNG
   RUNG wire#w1
      Coil( "Unit1.Em6.ControlNodes".visionUnit."step".transition[1001] )
   END_RUNG
   RUNG wire#w1
      Contact( "Unit1.Em6.ControlNodes".visionUnit."step".transition[1001] )
      { S7_Templates := "time_type := Time" } #statTonTimer[1001].TON(pt := #SeqNoDelayTime, et =>)
      Move(in := #JOB_10_STEP_11, out1 => "Unit1.Em6.ControlNodes".visionUnit.sequence.status.nextStep)
   END_RUNG
   // the same network as SCL:
   "Unit1.Em6.ControlNodes".visionUnit."step".action[1001] := ("Unit1.Em6.ControlNodes".visionUnit.sequence.status.currentStep = #JOB_10_STEP_01) AND "Unit1.Em6.ControlNodes".visionUnit.sequence.status.seqActive;
   "Unit1.Em6.ControlNodes".visionUnit."step".transition[1001] := ("Unit1.Em6.ControlNodes".visionUnit.sequence.status.currentStep = #JOB_10_STEP_01) AND "Unit1.Em6.ControlNodes".visionUnit.sequence.status.seqActive;
   #statTonTimer[1001].TON(IN := ("Unit1.Em6.ControlNodes".visionUnit.sequence.status.currentStep = #JOB_10_STEP_01) AND "Unit1.Em6.ControlNodes".visionUnit.sequence.status.seqActive AND "Unit1.Em6.ControlNodes".visionUnit."step".transition[1001],
                           PT := #SeqNoDelayTime);
   IF #statTonTimer[1001].Q THEN
       "Unit1.Em6.ControlNodes".visionUnit.sequence.status.nextStep := #JOB_10_STEP_11;
   END_IF;
END_REGION

REGION Network 22: Step[1011] : Vision Unit AxisZ WorkPos Command
   RUNG wire#powerrail
      { S7_Templates := "SrcType := DInt" } EQ_Contact(in1 := "Unit1.Em6.ControlNodes".visionUnit.sequence.status.currentStep, in2 := #JOB_10_STEP_11)
      Contact( "Unit1.Em6.ControlNodes".visionUnit.sequence.status.seqActive )
      wire#w1
      I_Contact( "Unit1.Em6.ControlNodes".cm.softcam.visionUnit.visionPos.inPos )
      Move(in := #VisionUnitAxisZVisionPos, out1 => "Unit1.Em6.ControlNodes".cmVisionUnitAxisZ.commands.selectSetPosition)
      Coil( "Unit1.Em6.ControlNodes".visionUnit."step".action[1011] )
   END_RUNG
   RUNG wire#w1
      Contact( "Unit1.Em6.ControlNodes".cm.softcam.visionUnit.visionPos.inPos )
      Coil( "Unit1.Em6.ControlNodes".visionUnit."step".transition[1011] )
   END_RUNG
   RUNG wire#w1
      Contact( "Unit1.Em6.ControlNodes".visionUnit."step".transition[1011] )
      { S7_Templates := "time_type := Time" } #statTonTimer[1011].TON(pt := #SeqDelayTime, et =>)
      Move(in := #JOB_10_STEP_21, out1 => "Unit1.Em6.ControlNodes".visionUnit.sequence.status.nextStep)
   END_RUNG
   // the same network as SCL:
   #_w1 := ("Unit1.Em6.ControlNodes".visionUnit.sequence.status.currentStep = #JOB_10_STEP_11) AND "Unit1.Em6.ControlNodes".visionUnit.sequence.status.seqActive;
   #_w2 := #_w1 AND NOT "Unit1.Em6.ControlNodes".cm.softcam.visionUnit.visionPos.inPos;
   IF #_w2 THEN
       "Unit1.Em6.ControlNodes".cmVisionUnitAxisZ.commands.selectSetPosition := #VisionUnitAxisZVisionPos;
   END_IF;
   "Unit1.Em6.ControlNodes".visionUnit."step".action[1011] := #_w2;
   "Unit1.Em6.ControlNodes".visionUnit."step".transition[1011] := #_w1 AND "Unit1.Em6.ControlNodes".cm.softcam.visionUnit.visionPos.inPos;
   #statTonTimer[1011].TON(IN := #_w1 AND "Unit1.Em6.ControlNodes".visionUnit."step".transition[1011],
                           PT := #SeqDelayTime);
   IF #statTonTimer[1011].Q THEN
       "Unit1.Em6.ControlNodes".visionUnit.sequence.status.nextStep := #JOB_10_STEP_21;
   END_IF;
END_REGION

REGION Network 23: Step[1021] : Vision Controller Trigger & QR Reader Trigger
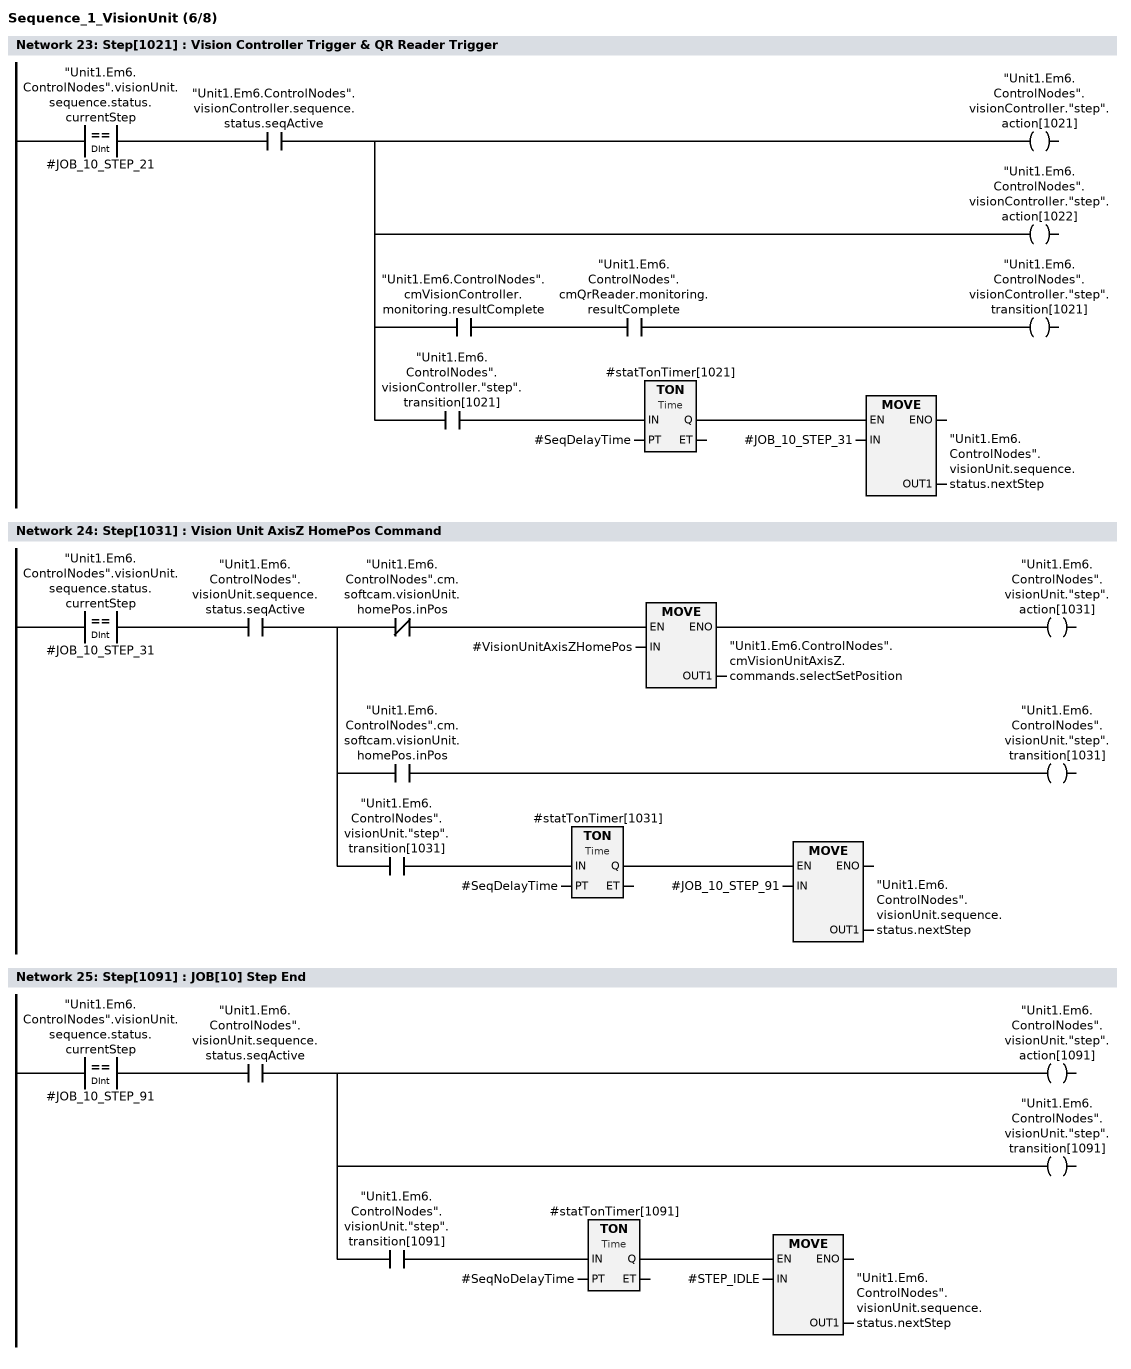
   RUNG wire#powerrail
      { S7_Templates := "SrcType := DInt" } EQ_Contact(in1 := "Unit1.Em6.ControlNodes".visionUnit.sequence.status.currentStep, in2 := #JOB_10_STEP_21)
      Contact( "Unit1.Em6.ControlNodes".visionController.sequence.status.seqActive )
      wire#w1
      Coil( "Unit1.Em6.ControlNodes".visionController."step".action[1021] )
   END_RUNG
   RUNG wire#w1
      Coil( "Unit1.Em6.ControlNodes".visionController."step".action[1022] )
   END_RUNG
   RUNG wire#w1
      Contact( "Unit1.Em6.ControlNodes".cmVisionController.monitoring.resultComplete )
      Contact( "Unit1.Em6.ControlNodes".cmQrReader.monitoring.resultComplete )
      Coil( "Unit1.Em6.ControlNodes".visionController."step".transition[1021] )
   END_RUNG
   RUNG wire#w1
      Contact( "Unit1.Em6.ControlNodes".visionController."step".transition[1021] )
      { S7_Templates := "time_type := Time" } #statTonTimer[1021].TON(pt := #SeqDelayTime, et =>)
      Move(in := #JOB_10_STEP_31, out1 => "Unit1.Em6.ControlNodes".visionUnit.sequence.status.nextStep)
   END_RUNG
   // the same network as SCL:
   "Unit1.Em6.ControlNodes".visionController."step".action[1021] := ("Unit1.Em6.ControlNodes".visionUnit.sequence.status.currentStep = #JOB_10_STEP_21) AND "Unit1.Em6.ControlNodes".visionController.sequence.status.seqActive;
   "Unit1.Em6.ControlNodes".visionController."step".action[1022] := ("Unit1.Em6.ControlNodes".visionUnit.sequence.status.currentStep = #JOB_10_STEP_21) AND "Unit1.Em6.ControlNodes".visionController.sequence.status.seqActive;
   "Unit1.Em6.ControlNodes".visionController."step".transition[1021] := ("Unit1.Em6.ControlNodes".visionUnit.sequence.status.currentStep = #JOB_10_STEP_21) AND "Unit1.Em6.ControlNodes".visionController.sequence.status.seqActive AND "Unit1.Em6.ControlNodes".cmVisionController.monitoring.resultComplete AND "Unit1.Em6.ControlNodes".cmQrReader.monitoring.resultComplete;
   #statTonTimer[1021].TON(IN := ("Unit1.Em6.ControlNodes".visionUnit.sequence.status.currentStep = #JOB_10_STEP_21) AND "Unit1.Em6.ControlNodes".visionController.sequence.status.seqActive AND "Unit1.Em6.ControlNodes".visionController."step".transition[1021],
                           PT := #SeqDelayTime);
   IF #statTonTimer[1021].Q THEN
       "Unit1.Em6.ControlNodes".visionUnit.sequence.status.nextStep := #JOB_10_STEP_31;
   END_IF;
END_REGION

REGION Network 24: Step[1031] : Vision Unit AxisZ HomePos Command
   RUNG wire#powerrail
      { S7_Templates := "SrcType := DInt" } EQ_Contact(in1 := "Unit1.Em6.ControlNodes".visionUnit.sequence.status.currentStep, in2 := #JOB_10_STEP_31)
      Contact( "Unit1.Em6.ControlNodes".visionUnit.sequence.status.seqActive )
      wire#w1
      I_Contact( "Unit1.Em6.ControlNodes".cm.softcam.visionUnit.homePos.inPos )
      Move(in := #VisionUnitAxisZHomePos, out1 => "Unit1.Em6.ControlNodes".cmVisionUnitAxisZ.commands.selectSetPosition)
      Coil( "Unit1.Em6.ControlNodes".visionUnit."step".action[1031] )
   END_RUNG
   RUNG wire#w1
      Contact( "Unit1.Em6.ControlNodes".cm.softcam.visionUnit.homePos.inPos )
      Coil( "Unit1.Em6.ControlNodes".visionUnit."step".transition[1031] )
   END_RUNG
   RUNG wire#w1
      Contact( "Unit1.Em6.ControlNodes".visionUnit."step".transition[1031] )
      { S7_Templates := "time_type := Time" } #statTonTimer[1031].TON(pt := #SeqDelayTime, et =>)
      Move(in := #JOB_10_STEP_91, out1 => "Unit1.Em6.ControlNodes".visionUnit.sequence.status.nextStep)
   END_RUNG
   // the same network as SCL:
   #_w1 := ("Unit1.Em6.ControlNodes".visionUnit.sequence.status.currentStep = #JOB_10_STEP_31) AND "Unit1.Em6.ControlNodes".visionUnit.sequence.status.seqActive;
   #_w2 := #_w1 AND NOT "Unit1.Em6.ControlNodes".cm.softcam.visionUnit.homePos.inPos;
   IF #_w2 THEN
       "Unit1.Em6.ControlNodes".cmVisionUnitAxisZ.commands.selectSetPosition := #VisionUnitAxisZHomePos;
   END_IF;
   "Unit1.Em6.ControlNodes".visionUnit."step".action[1031] := #_w2;
   "Unit1.Em6.ControlNodes".visionUnit."step".transition[1031] := #_w1 AND "Unit1.Em6.ControlNodes".cm.softcam.visionUnit.homePos.inPos;
   #statTonTimer[1031].TON(IN := #_w1 AND "Unit1.Em6.ControlNodes".visionUnit."step".transition[1031],
                           PT := #SeqDelayTime);
   IF #statTonTimer[1031].Q THEN
       "Unit1.Em6.ControlNodes".visionUnit.sequence.status.nextStep := #JOB_10_STEP_91;
   END_IF;
END_REGION

REGION Network 25: Step[1091] : JOB[10] Step End
   RUNG wire#powerrail
      { S7_Templates := "SrcType := DInt" } EQ_Contact(in1 := "Unit1.Em6.ControlNodes".visionUnit.sequence.status.currentStep, in2 := #JOB_10_STEP_91)
      Contact( "Unit1.Em6.ControlNodes".visionUnit.sequence.status.seqActive )
      wire#w1
      Coil( "Unit1.Em6.ControlNodes".visionUnit."step".action[1091] )
   END_RUNG
   RUNG wire#w1
      Coil( "Unit1.Em6.ControlNodes".visionUnit."step".transition[1091] )
   END_RUNG
   RUNG wire#w1
      Contact( "Unit1.Em6.ControlNodes".visionUnit."step".transition[1091] )
      { S7_Templates := "time_type := Time" } #statTonTimer[1091].TON(pt := #SeqNoDelayTime, et =>)
      Move(in := #STEP_IDLE, out1 => "Unit1.Em6.ControlNodes".visionUnit.sequence.status.nextStep)
   END_RUNG
   // the same network as SCL:
   "Unit1.Em6.ControlNodes".visionUnit."step".action[1091] := ("Unit1.Em6.ControlNodes".visionUnit.sequence.status.currentStep = #JOB_10_STEP_91) AND "Unit1.Em6.ControlNodes".visionUnit.sequence.status.seqActive;
   "Unit1.Em6.ControlNodes".visionUnit."step".transition[1091] := ("Unit1.Em6.ControlNodes".visionUnit.sequence.status.currentStep = #JOB_10_STEP_91) AND "Unit1.Em6.ControlNodes".visionUnit.sequence.status.seqActive;
   #statTonTimer[1091].TON(IN := ("Unit1.Em6.ControlNodes".visionUnit.sequence.status.currentStep = #JOB_10_STEP_91) AND "Unit1.Em6.ControlNodes".visionUnit.sequence.status.seqActive AND "Unit1.Em6.ControlNodes".visionUnit."step".transition[1091],
                           PT := #SeqNoDelayTime);
   IF #statTonTimer[1091].Q THEN
       "Unit1.Em6.ControlNodes".visionUnit.sequence.status.nextStep := #STEP_IDLE;
   END_IF;
END_REGION

REGION Network 26: *************** IMMEDIATE STOP ****************
END_REGION

REGION Network 27: Immediate Stop
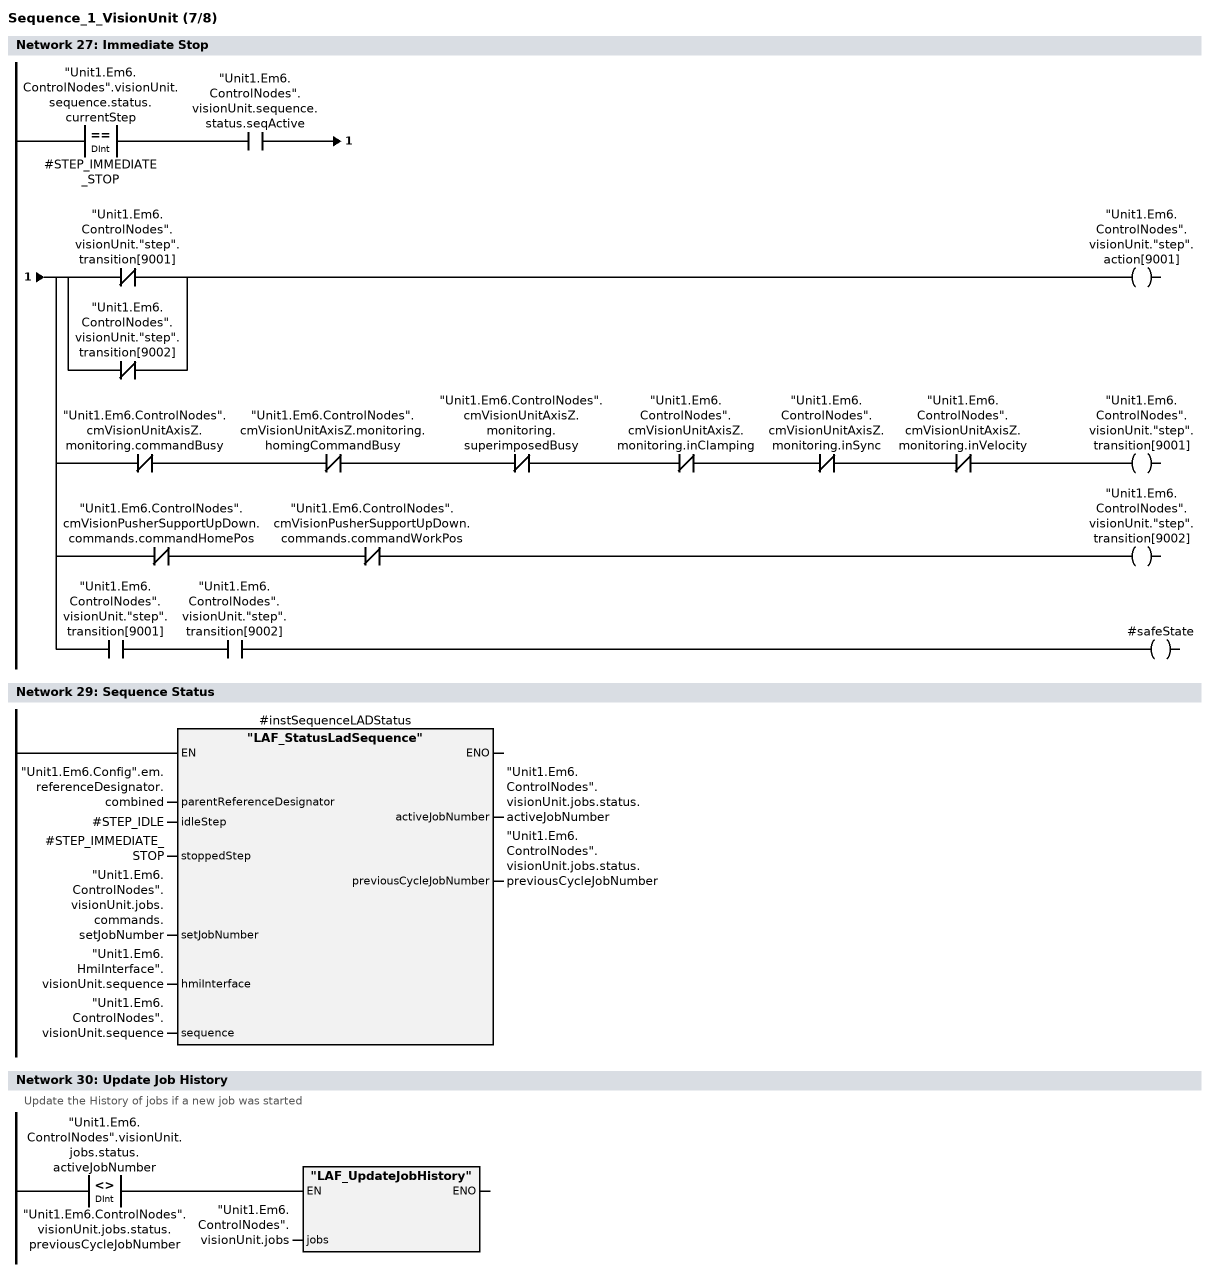
   RUNG wire#powerrail
      { S7_Templates := "SrcType := DInt" } EQ_Contact(in1 := "Unit1.Em6.ControlNodes".visionUnit.sequence.status.currentStep, in2 := #STEP_IMMEDIATE_STOP)
      Contact( "Unit1.Em6.ControlNodes".visionUnit.sequence.status.seqActive )
      wire#w1
      I_Contact( "Unit1.Em6.ControlNodes".visionUnit."step".transition[9001] )
      wire#w2
      Coil( "Unit1.Em6.ControlNodes".visionUnit."step".action[9001] )
   END_RUNG
   RUNG wire#w1
      I_Contact( "Unit1.Em6.ControlNodes".visionUnit."step".transition[9002] )
   END_RUNG wire#w2
   RUNG wire#w1
      I_Contact( "Unit1.Em6.ControlNodes".cmVisionUnitAxisZ.monitoring.commandBusy )
      I_Contact( "Unit1.Em6.ControlNodes".cmVisionUnitAxisZ.monitoring.homingCommandBusy )
      I_Contact( "Unit1.Em6.ControlNodes".cmVisionUnitAxisZ.monitoring.superimposedBusy )
      I_Contact( "Unit1.Em6.ControlNodes".cmVisionUnitAxisZ.monitoring.inClamping )
      I_Contact( "Unit1.Em6.ControlNodes".cmVisionUnitAxisZ.monitoring.inSync )
      I_Contact( "Unit1.Em6.ControlNodes".cmVisionUnitAxisZ.monitoring.inVelocity )
      Coil( "Unit1.Em6.ControlNodes".visionUnit."step".transition[9001] )
   END_RUNG
   RUNG wire#w1
      I_Contact( "Unit1.Em6.ControlNodes".cmVisionPusherSupportUpDown.commands.commandHomePos )
      I_Contact( "Unit1.Em6.ControlNodes".cmVisionPusherSupportUpDown.commands.commandWorkPos )
      Coil( "Unit1.Em6.ControlNodes".visionUnit."step".transition[9002] )
   END_RUNG
   RUNG wire#w1
      Contact( "Unit1.Em6.ControlNodes".visionUnit."step".transition[9001] )
      Contact( "Unit1.Em6.ControlNodes".visionUnit."step".transition[9002] )
      Coil( #safeState )
   END_RUNG
   // the same network as SCL:
   #_w1 := ("Unit1.Em6.ControlNodes".visionUnit.sequence.status.currentStep = #STEP_IMMEDIATE_STOP) AND "Unit1.Em6.ControlNodes".visionUnit.sequence.status.seqActive;
   "Unit1.Em6.ControlNodes".visionUnit."step".action[9001] := #_w1 AND (NOT "Unit1.Em6.ControlNodes".visionUnit."step".transition[9001] OR NOT "Unit1.Em6.ControlNodes".visionUnit."step".transition[9002]);
   "Unit1.Em6.ControlNodes".visionUnit."step".transition[9001] := #_w1 AND NOT "Unit1.Em6.ControlNodes".cmVisionUnitAxisZ.monitoring.commandBusy AND NOT "Unit1.Em6.ControlNodes".cmVisionUnitAxisZ.monitoring.homingCommandBusy AND NOT "Unit1.Em6.ControlNodes".cmVisionUnitAxisZ.monitoring.superimposedBusy AND NOT "Unit1.Em6.ControlNodes".cmVisionUnitAxisZ.monitoring.inClamping AND NOT "Unit1.Em6.ControlNodes".cmVisionUnitAxisZ.monitoring.inSync AND NOT "Unit1.Em6.ControlNodes".cmVisionUnitAxisZ.monitoring.inVelocity;
   "Unit1.Em6.ControlNodes".visionUnit."step".transition[9002] := #_w1 AND NOT "Unit1.Em6.ControlNodes".cmVisionPusherSupportUpDown.commands.commandHomePos AND NOT "Unit1.Em6.ControlNodes".cmVisionPusherSupportUpDown.commands.commandWorkPos;
   #safeState := #_w1 AND "Unit1.Em6.ControlNodes".visionUnit."step".transition[9001] AND "Unit1.Em6.ControlNodes".visionUnit."step".transition[9002];
END_REGION

REGION Network 28: *************** STATUS **********************
END_REGION

REGION Network 29: Sequence Status
   RUNG wire#powerrail
      #instSequenceLADStatus(parentReferenceDesignator := "Unit1.Em6.Config".em.referenceDesignator.combined, idleStep := #STEP_IDLE, stoppedStep := #STEP_IMMEDIATE_STOP, setJobNumber := "Unit1.Em6.ControlNodes".visionUnit.jobs.commands.setJobNumber, hmiInterface := "Unit1.Em6.HmiInterface".visionUnit.sequence, sequence := "Unit1.Em6.ControlNodes".visionUnit.sequence, activeJobNumber => "Unit1.Em6.ControlNodes".visionUnit.jobs.status.activeJobNumber, previousCycleJobNumber => "Unit1.Em6.ControlNodes".visionUnit.jobs.status.previousCycleJobNumber)
   END_RUNG
   // the same network as SCL:
   #instSequenceLADStatus(parentReferenceDesignator := "Unit1.Em6.Config".em.referenceDesignator.combined,   // "LAF_StatusLadSequence"
                          idleStep := #STEP_IDLE,
                          stoppedStep := #STEP_IMMEDIATE_STOP,
                          setJobNumber := "Unit1.Em6.ControlNodes".visionUnit.jobs.commands.setJobNumber,
                          hmiInterface := "Unit1.Em6.HmiInterface".visionUnit.sequence,
                          sequence := "Unit1.Em6.ControlNodes".visionUnit.sequence,
                          activeJobNumber => "Unit1.Em6.ControlNodes".visionUnit.jobs.status.activeJobNumber,
                          previousCycleJobNumber => "Unit1.Em6.ControlNodes".visionUnit.jobs.status.previousCycleJobNumber);
END_REGION

REGION Network 30: Update Job History
   // Update the History of jobs if a new job was started
   RUNG wire#powerrail
      { S7_Templates := "SrcType := DInt" } NE_Contact(in1 := "Unit1.Em6.ControlNodes".visionUnit.jobs.status.activeJobNumber, in2 := "Unit1.Em6.ControlNodes".visionUnit.jobs.status.previousCycleJobNumber)
      "LAF_UpdateJobHistory"(jobs := "Unit1.Em6.ControlNodes".visionUnit.jobs)
   END_RUNG
   // the same network as SCL:
   IF "Unit1.Em6.ControlNodes".visionUnit.jobs.status.activeJobNumber <> "Unit1.Em6.ControlNodes".visionUnit.jobs.status.previousCycleJobNumber THEN
       "LAF_UpdateJobHistory"(jobs := "Unit1.Em6.ControlNodes".visionUnit.jobs);
   END_IF;
END_REGION

REGION Network 31: Output steps as String
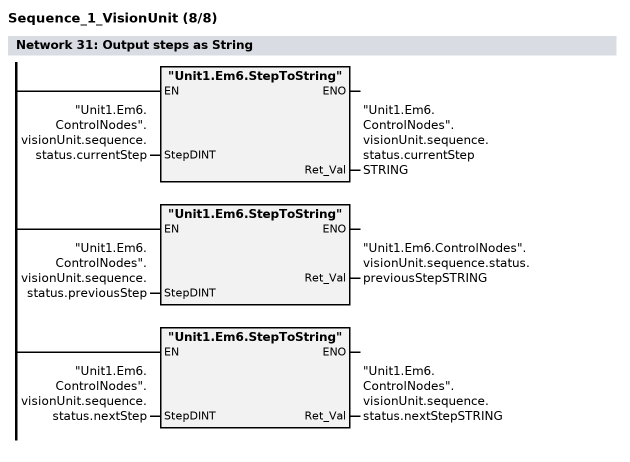
   RUNG wire#powerrail
      "Unit1.Em6.StepToString"(StepDINT := "Unit1.Em6.ControlNodes".visionUnit.sequence.status.currentStep, Ret_Val => "Unit1.Em6.ControlNodes".visionUnit.sequence.status.currentStepSTRING)
   END_RUNG
   RUNG wire#powerrail
      "Unit1.Em6.StepToString"(StepDINT := "Unit1.Em6.ControlNodes".visionUnit.sequence.status.previousStep, Ret_Val => "Unit1.Em6.ControlNodes".visionUnit.sequence.status.previousStepSTRING)
   END_RUNG
   RUNG wire#powerrail
      "Unit1.Em6.StepToString"(StepDINT := "Unit1.Em6.ControlNodes".visionUnit.sequence.status.nextStep, Ret_Val => "Unit1.Em6.ControlNodes".visionUnit.sequence.status.nextStepSTRING)
   END_RUNG
   // the same network as SCL:
   "Unit1.Em6.ControlNodes".visionUnit.sequence.status.currentStepSTRING := "Unit1.Em6.StepToString"(StepDINT := "Unit1.Em6.ControlNodes".visionUnit.sequence.status.currentStep);
   "Unit1.Em6.ControlNodes".visionUnit.sequence.status.previousStepSTRING := "Unit1.Em6.StepToString"(StepDINT := "Unit1.Em6.ControlNodes".visionUnit.sequence.status.previousStep);
   "Unit1.Em6.ControlNodes".visionUnit.sequence.status.nextStepSTRING := "Unit1.Em6.StepToString"(StepDINT := "Unit1.Em6.ControlNodes".visionUnit.sequence.status.nextStep);
END_REGION
END_FUNCTION_BLOCK
